PROGRAM P_Demo_PHUGE_TO_HUGE
VAR
    hRealValue           : HUGE; // 模拟 wire 缓冲区中的 HUGE 字段
    pHUGEField           : POINTER TO HUGE; // 业务侧先算好的字段地址（ADR 或 pBase+nOff）
    bExtractField        : BOOL; // 在线置 TRUE 触发一次解析
    hRealValue_extracted : HUGE; // 解析后的副本，供业务逻辑使用
END_VAR

// ============================================================
// Tc2_Utilities.PHUGE_TO_HUGE 演示程序（FUNCTION）
// ============================================================
// 场景：从一段二进制 wire 缓冲区里按偏移取 HUGE 字段（Modbus/CAN/ADS Raw）。
// 价值：替代手写 pField + nOff + ^ 指针算术；一次调用取值，少打错符号。
// 验证：在线写 hRealValue := 示例值；bExtractField := TRUE；
//       下一周期 hRealValue_extracted 应等于 hRealValue。
// ============================================================

// 业务代码通常已经算好字段地址（pBase + 协议偏移）；演示用 ADR 等价
pHUGEField := ADR(hRealValue);

IF bExtractField AND pHUGEField <> 0 THEN
    // 单次完整调用：避免手写 ^ 解引用，统一风格便于和字节序转换串联
    hRealValue_extracted := PHUGE_TO_HUGE(pHUGEField);
    bExtractField := FALSE;
END_IF;

END_PROGRAM

(* stored: Version 1.1.0.1, ProductVersion 3.1.4024.5
   POU P_Demo_PHUGE_TO_HUGE: Id {d8e0a02c-b890-5db9-822b-87cd9d62e81f}, SpecialFunc None *)
